{attribute addProperty BoxType "EPP2338-0001-0016"}
{attribute addProperty Id "ChannelAT %I*ARRAY[0..7] OF Channel_E4AEF59E6480Channel_1AT %Q*ARRAY[0..7] OF Channel_7F374EB06480WcStateAT %I*WcState_F855686C1620InfoDataAT %I*InfoData_192954DE1620"}
{attribute addProperty CRC "2833668530"}
{attribute addProperty SizeInBites "160"}
{attribute addProperty SizeInBytes "20"}
TYPE EPP2338_6598BC39 :
STRUCT
	{attribute addProperty Name "Channel"}
	Channel : ARRAY[0..7] OF Channel_E4AEF59E;
	{attribute addProperty Name "Channel_1"}
	Channel_1 : ARRAY[0..7] OF Channel_7F374EB0;
	{attribute addProperty Name "WcState"}
	WcState : WcState_F855686C;
	{attribute addProperty Name "InfoData"}
	InfoData : InfoData_192954DE;
END_STRUCT
END_TYPE

(* stored: Version 1.2.0.0, ProductVersion 3.1.4024.9
   DUT EPP2338_6598BC39: Id {04c50c9f-26cd-4525-bf83-dc1a0f7554ca} *)
